{attribute 'linkalways'} 
{attribute 'no_explicit_call' := 'This FB is a CLASS and must be accessed using methods or properties'}
{attribute 'enable_dynamic_creation'}
FUNCTION_BLOCK _ETcVnSvmSgdClassifierMarginType EXTENDS EnumDatatypeBase
VAR
	localData : ETcVnSvmSgdClassifierMarginType;
	activeData : REFERENCE TO ETcVnSvmSgdClassifierMarginType;
	enumBaseDatatype : _DINT(localData);
END_VAR

METHOD PRIVATE AddLocalEnumeration
VAR_INPUT
	Enumeration : T_MAXSTRING;
	Value : ETcVnSvmSgdClassifierMarginType;
END_VAR
AddEnumeration(Enumeration, Value);
END_METHOD

PROPERTY PUBLIC Address : PVOID
GET
Address := ADR(activeData);
END_GET
END_PROPERTY

METHOD PUBLIC ClearReference
VAR_INPUT
END_VAR
activeData REF= localData;
SetBaseDatatypeReference();
END_METHOD

METHOD PUBLIC Clone : I_Datatype
VAR
    pClone : POINTER TO _ETcVnSvmSgdClassifierMarginType;
END_VAR
pClone := __NEW(_ETcVnSvmSgdClassifierMarginType(InitialValue := Value));
Clone := pClone^;
END_METHOD

METHOD FB_init : BOOL
VAR_INPUT
	bInitRetains : BOOL; // if TRUE, the retain variables are initialized (warm start / cold start)
	bInCopyCode : BOOL;  // if TRUE, the instance afterwards gets moved into the copy code (online change)
	InitialValue : ETcVnSvmSgdClassifierMarginType;
END_VAR
localData := InitialValue;
AddBaseDatatype(enumBaseDatatype);
ClearReference();

AddLocalEnumeration('TCVN_SSCMT_SOFT_MARGIN', ETcVnSvmSgdClassifierMarginType.TCVN_SSCMT_SOFT_MARGIN);
AddLocalEnumeration('TCVN_SSCMT_HARD_MARGIN', ETcVnSvmSgdClassifierMarginType.TCVN_SSCMT_HARD_MARGIN);
END_METHOD

PROPERTY PUBLIC Identifier : T_MAXSTRING
GET
Identifier := 'ETcVnSvmSgdClassifierMarginType';
END_GET
END_PROPERTY

METHOD IsEnumeratorValueEqual : BOOL
VAR_INPUT
	Enumerator : I_KeyValueForwardEnumerator;
END_VAR
VAR
	storedValue : ETcVnSvmSgdClassifierMarginType;
END_VAR
IF NOT Enumerator.TryGet(storedValue) THEN
	RETURN;
END_IF

IsEnumeratorValueEqual := storedValue = activeData;
END_METHOD

METHOD PUBLIC MakeReferenceTo
VAR_INPUT
	ReferenceTarget : REFERENCE TO ETcVnSvmSgdClassifierMarginType;
END_VAR
activeData REF= ReferenceTarget;
SetBaseDatatypeReference();
END_METHOD

METHOD PROTECTED SetBaseDatatypeReference
VAR_INPUT
END_VAR
enumBaseDatatype.MakeReferenceTo(activeData);
END_METHOD

PROPERTY PUBLIC Size : UDINT
GET
Size := SIZEOF(activeData);
END_GET
END_PROPERTY

METHOD TryMakeReferenceTo : BOOL
VAR_INPUT
	Target : I_Datatype;
END_VAR
VAR
	targetAsEnum : I_EnumDatatype;
	pTargetData : POINTER TO ETcVnSvmSgdClassifierMarginType;
END_VAR
IF NOT Target.TryResolveAsEnumDatatype(targetAsEnum) THEN
	RETURN;
END_IF

IF targetAsEnum.Identifier <> Identifier THEN
	RETURN;
END_IF

pTargetData := Target.Address;
activeData REF= pTargetData^;
SetBaseDatatypeReference();
TryMakeReferenceTo := TRUE;
END_METHOD

PROPERTY PUBLIC Value : ETcVnSvmSgdClassifierMarginType
GET
Value := activeData;
END_GET
SET
activeData := Value;
END_SET
END_PROPERTY

END_FUNCTION_BLOCK

(* stored: Version 1.1.0.1, ProductVersion 3.1.4024.12
   POU _ETcVnSvmSgdClassifierMarginType: Id {d180a67f-1605-4a99-800f-463cc0d2cfa8}, SpecialFunc None
   Folder Constructor: Id {d0c33d22-a235-46d2-a0b5-955510c1486f}
   Folder Private: Id {e6b2d333-aef0-4f36-9b10-e0e35edc91a6}
   Folder Protected: Id {805a6009-1130-4a18-8231-b5903ebc8b3f}
   Method AddLocalEnumeration: Id {333c0e8e-2cc9-4a5d-aa3d-621aa729feb1}
   Property Address: Id {537b2182-09c9-460f-97c5-1bfb73e1f3f5}
   Get Get: Id {c16398ad-59fc-41d6-9745-5524eceb275a}
   Method ClearReference: Id {03a0d5de-8f01-4383-ac11-9e6581bc79b4}
   Method Clone: Id {c9fdfdec-4f4b-4ae2-a606-04bf3d3301d6}
   Method FB_init: Id {47c3d53d-e6b7-4cc2-9e0a-9a3e44ddf8c9}
   Property Identifier: Id {e58dfa58-f135-4328-9346-665a87f22228}
   Get Get: Id {b718167f-8e96-46c9-8170-c9344a2fe327}
   Method IsEnumeratorValueEqual: Id {f9dd82b6-593e-4609-807b-c17b053e538e}
   Method MakeReferenceTo: Id {11e01060-0037-4074-9443-56e4e38b4a05}
   Method SetBaseDatatypeReference: Id {e4c81e4b-5dec-4c55-8b6b-4e73969e15e7}
   Property Size: Id {859501b2-91e3-47bc-85a5-65eff71cca46}
   Get Get: Id {b34a20e4-f3dc-4345-ba4d-8794eace49b4}
   Method TryMakeReferenceTo: Id {4bc917f3-6247-4484-bcf9-de6e223ffcf5}
   Property Value: Id {feb734a4-d6ad-4fad-9ee4-38f7c31353d2}
   Get Get: Id {e9419383-b4dc-4c7a-8770-b95b585fdcd4}
   Set Set: Id {89528121-f23f-4c28-be9e-cde3c234b5cd} *)
